{attribute 'TcGenerated'}
{attribute 'no-analysis'}
{attribute 'linkalways'}
// This function has been automatically generated from the project information.
VAR_GLOBAL CONSTANT
	{attribute 'const_non_replaced'}
	stLibVersion_Tk_MachineControl : ST_LibVersion := (iMajor := 0, iMinor := 0, iBuild := 3, iRevision := 1, nFlags := 0, sVersion := '0.0.3.1');
END_VAR

(* stored: Version 1.1.0.1
   GVL Global_Version: Id {60559a3d-45b2-4650-932c-d4127b87839b} *)
